(* Initialise les devices *)
FUNCTION_BLOCK HardwareManager
VAR_INPUT			
END_VAR
VAR_OUTPUT
END_VAR
VAR	
	{attribute 'OPC.UA.DA' := '0'}
	{attribute 'OPC.UA.DA.StructuredType' := '0'}
	ProcessModulesConfig : ProcessModulesConfig;	

	{attribute 'OPC.UA.DA' := '0'}
	{attribute 'OPC.UA.DA.StructuredType' := '0'}
	CalibratePMsConfig : CalibratePMsConfig;
	
	{region "PMs" } 	
	
	{attribute 'OPC.UA.DA' := '1'}
	{attribute 'OPC.UA.DA.StructuredType' := '1'}	 
	Lightspeed : Lightspeed(Config := ProcessModulesConfig.LightspeedConfig, CalibrateConfig := CalibratePMsConfig.LsCalibrateConfig);

	{attribute 'OPC.UA.DA' := '1'}
	{attribute 'OPC.UA.DA.StructuredType' := '1'}			
	Psd : Psd(Config := ProcessModulesConfig.PsdConfig);
		
	{attribute 'OPC.UA.DA' := '1'}
	{attribute 'OPC.UA.DA.StructuredType' := '1'}	 
	Nst : Nst(Config := ProcessModulesConfig.NstConfig);
 
	{attribute 'OPC.UA.DA' := '1'}
	{attribute 'OPC.UA.DA.StructuredType' := '1'}	 
	PhotoLum : PhotoLum(Config := ProcessModulesConfig.PhotoLumConfig);
		   
	{endregion}
					  	
	{attribute 'hide'}  
	_initializedHardware : BOOL;
	{attribute 'hide'}  
	_initializedCalibrate : BOOL ; //:= TRUE;  TODO pourquoi la calibration de la NST pose problème ? 
	
	{attribute 'OPC.UA.DA' := '0'}
	_xmlCalibrate : TXml;
	{attribute 'OPC.UA.DA' := '0'}
	_xmlHardware : TXml;
	{attribute 'OPC.UA.DA' := '0'}
	_logger : Logger;
	{attribute 'OPC.UA.DA' := '0'}
	_message : StringBuilder;
		
END_VAR

IF NOT _initializedCalibrate AND NOT _xmlCalibrate.DeserialisationOperation.Error THEN  
	InitCalibrate();	
END_IF	

IF _initializedCalibrate AND NOT _initializedHardware AND NOT 
	_xmlHardware.DeserialisationOperation.Error THEN
	
	InitHardware();
END_IF

IF  _initializedHardware AND _initializedCalibrate THEN
	IF ProcessModulesConfig.LightspeedConfig.IsEnabled THEN
		Lightspeed();	
	END_IF

	IF ProcessModulesConfig.PsdConfig.IsEnabled THEN
		Psd();	
	END_IF		
	
	IF ProcessModulesConfig.NstConfig.IsEnabled THEN
		Nst();	
	END_IF
	
	IF ProcessModulesConfig.PhotoLumConfig.IsEnabled THEN
		PhotoLum();	
	END_IF
END_IF

ACTION CalibrateDeserialize:
_xmlCalibrate(FilePath := GlobalConfig.AppConfig.CalibrateConfig.CalibratePath, 
	 		  XPath := GlobalConfig.AppConfig.CalibrateConfig.CalibrateHeaderNodeXml,  
	 		  AddHeaderNodeXml := ADR(CalibratePMsConfig), 
	 		  SizeOfHeaderNodeXml := SIZEOF(CalibratePMsConfig));
END_ACTION

ACTION HardwareDeserialize:
_xmlHardware(FilePath := GlobalConfig.AppConfig.LogConfig.LogFileConfigPath, 
	 		 XPath := GlobalConfig.AppConfig.LogConfig.HeaderNodeXml, 
	 		 AddHeaderNodeXml := ADR(ProcessModulesConfig), 
	 		 SizeOfHeaderNodeXml := SIZEOF(ProcessModulesConfig));
END_ACTION

METHOD InitCalibrate : BOOL
VAR_INPUT
END_VAR

IF _xmlCalibrate.DeserialisationOperation.Ready THEN
	_logger.Information(_message.Reset().Append('Loading calibrate configuration from ').
						    		 	 Append(TO_STRING(GlobalConfig.AppConfig.CalibrateConfig.CalibratePath)).ToString());
END_IF;	

_xmlCalibrate.DeserialisationOperation.Start();
CalibrateDeserialize();
	
IF _xmlCalibrate.DeserialisationOperation.Done THEN
	_logger.Information('Calibrate configuration loading done');	
	_xmlCalibrate.DeserialisationOperation.SetReady();		
	
	_initializedCalibrate := TRUE;
END_IF
 
IF _xmlCalibrate.DeserialisationOperation.Error THEN	
	_logger.Error('Calibrate load initialization error '); 
	_xmlCalibrate.SetError(_xmlCalibrate.DeserialisationOperation.ErrorId);
	
	_initializedCalibrate := FALSE;
END_IF
END_METHOD

METHOD PRIVATE InitHardware : BOOL
VAR_INPUT
END_VAR
VAR
END_VAR

IF _xmlHardware.DeserialisationOperation.Ready THEN
	_logger.Information(_message.Reset().Append('Loading hardware configuration from ').
						    		 	 Append(TO_STRING(GlobalConfig.AppConfig.LogConfig.LogFileConfigPath)).ToString());
END_IF;	

_xmlHardware.DeserialisationOperation.Start();
HardwareDeserialize();
	
IF _xmlHardware.DeserialisationOperation.Done THEN
	_logger.Information('Hardware configuration loading done');	
	_xmlHardware.DeserialisationOperation.SetReady();	
	
	// Load PMs
	IF ProcessModulesConfig.LightspeedConfig.IsEnabled THEN
		InitializeLightspeed();	
	END_IF
	
	IF ProcessModulesConfig.PsdConfig.IsEnabled THEN
		InitializePsd();	
	END_IF
	
	IF ProcessModulesConfig.NstConfig.IsEnabled THEN
		InitializeNst();	
	END_IF
	
	IF ProcessModulesConfig.PhotoLumConfig.IsEnabled THEN
		InitializePhotoLum();	
	END_IF
	
	_initializedHardware := TRUE;
END_IF
 
IF _xmlHardware.DeserialisationOperation.Error THEN	
	_logger.Error('Hardware load initialization error'); 
	_xmlHardware.SetError(_xmlHardware.DeserialisationOperation.ErrorId);
	
	_initializedHardware := FALSE;
END_IF
END_METHOD

METHOD InitializeLightspeed 
VAR_INPUT
END_VAR
Lightspeed.FB_init(FALSE, FALSE, Config := ProcessModulesConfig.LightspeedConfig, CalibrateConfig := CalibratePMsConfig.LsCalibrateConfig);
END_METHOD

METHOD InitializeNst 
VAR_INPUT
END_VAR
Nst.FB_init(FALSE, FALSE, Config := ProcessModulesConfig.NstConfig);
END_METHOD

METHOD InitializePhotoLum 
VAR_INPUT
END_VAR
PhotoLum.FB_init(FALSE, FALSE, Config := ProcessModulesConfig.PhotoLumConfig);
END_METHOD

METHOD InitializePsd 
VAR_INPUT
END_VAR
Psd.FB_init(FALSE, FALSE, Config := ProcessModulesConfig.PsdConfig);
END_METHOD

END_FUNCTION_BLOCK

(* stored: Version 1.1.0.1, ProductVersion 3.1.4024.12
   POU HardwareManager: Id {ed1eb7f5-2388-478b-891a-ab4f555591e3}, SpecialFunc None
   Action CalibrateDeserialize: Id {ed4d1625-f14d-4adf-9ddf-2ff25d88473c}
   Action HardwareDeserialize: Id {22c988d8-5cfe-4101-8a36-15d886901392}
   Method InitCalibrate: Id {a7eda3c5-c98e-4ce3-8fde-31673d528673}
   Method InitHardware: Id {4424e5ee-6b36-4882-aad1-846b130fc691}
   Method InitializeLightspeed: Id {fa44c0d2-38dc-401a-8f50-bd9ed9c3ea9a}
   Method InitializeNst: Id {912766b4-2c2b-45f7-b159-e15aae0130ad}
   Method InitializePhotoLum: Id {c6be157a-b300-48e3-be58-d652e551a068}
   Method InitializePsd: Id {fd730ddf-3852-46c6-8999-809dd93cc4be} *)
